TEXTLIST TL_E_CTRL_MOVER
  0 = 'MOVER_NULL'
  1 = 'MOVER_ENABLE'
  2 = 'MOVER_DISABLE'
  3 = 'MOVER_MOVE_TO_POS_CA'
  4 = 'MOVER_SEND_TO_POS_CA'
  5 = 'MOVER_HALT'
  6 = 'MOVER_GEAR_IN'
  7 = 'MOVER_GEAR_IN_POS_CA'
  8 = 'MOVER_GEAR_OUT'
  9 = 'MOVER_RESET'
   = ''
END_TEXTLIST

(* stored: Version 1.1.0.1, ProductVersion 3.1.4024.12
   TextList TL_E_CTRL_MOVER: Id {9b6b6994-12d1-49aa-a062-db5b553bf9be} *)
